// SIMATIC S7-200 project (STEP 7-Micro/WIN), CPU 221 REL 01.10

SYMBOL_TABLE USER1
S_tar            I0.0
S_top            I0.1
Den_1            Q0.0
Den_2            Q0.1
Den_3            Q0.2
Den_4            Q0.3
Den_5            Q0.4
END_SYMBOL_TABLE

ORGANIZATION_BLOCK MAIN:OB1
TITLE=PROGRAM COMMENTS
BEGIN
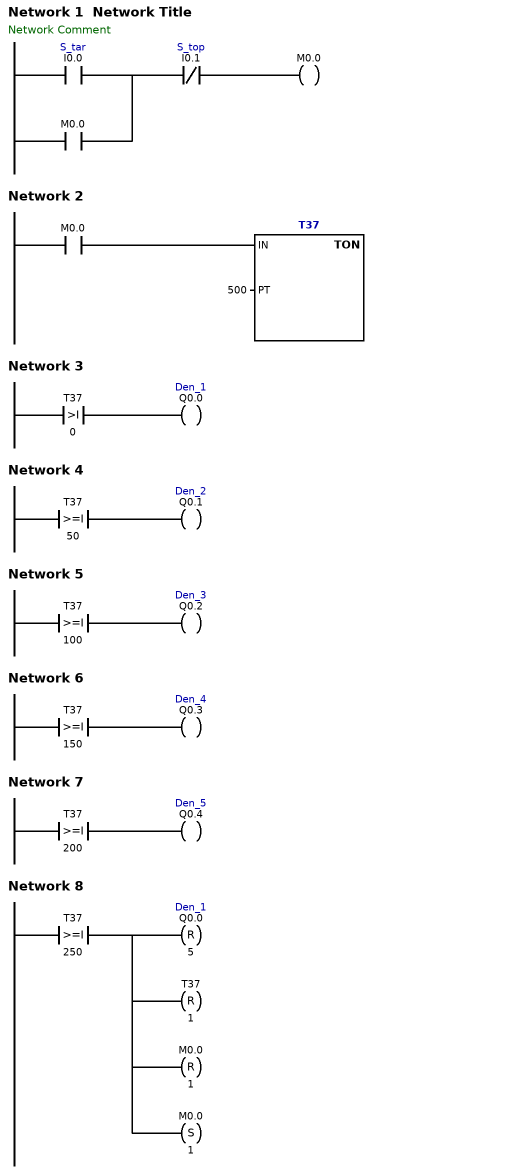
Network 1 // Network Title
// Network Comment
LD     S_tar:I0.0
O      M0.0
AN     S_top:I0.1
=      M0.0
Network 2
LD     M0.0
TON    T37, 500
Network 3
LDW>   T37, 0
=      Den_1:Q0.0
Network 4
LDW>=  T37, 50
=      Den_2:Q0.1
Network 5
LDW>=  T37, 100
=      Den_3:Q0.2
Network 6
LDW>=  T37, 150
=      Den_4:Q0.3
Network 7
LDW>=  T37, 200
=      Den_5:Q0.4
Network 8
LDW>=  T37, 250
R      Den_1:Q0.0, 5
R      T37, 1
R      M0.0, 1
S      M0.0, 1
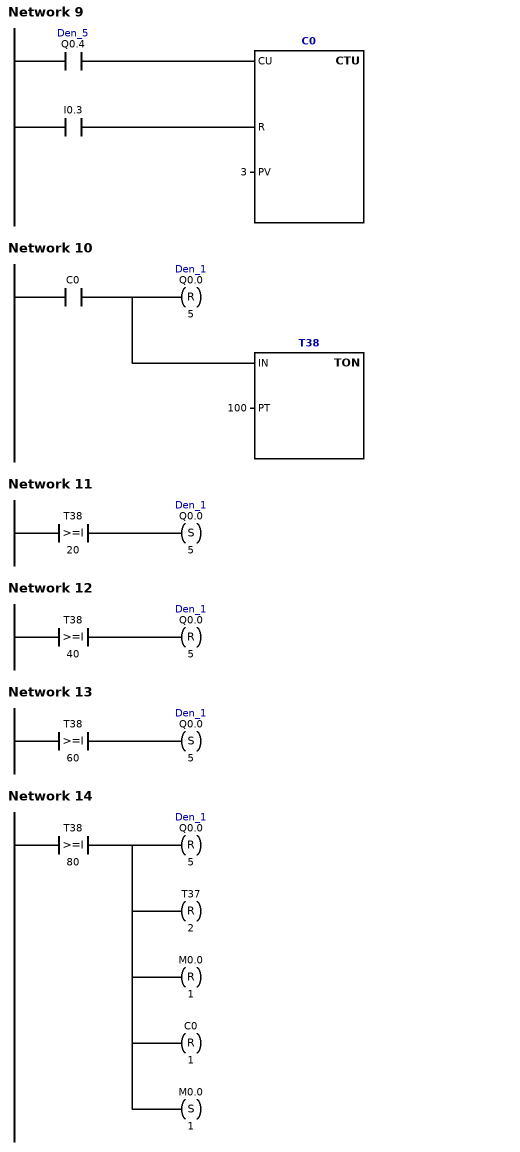
Network 9
LD     Den_5:Q0.4
LD     I0.3
CTU    C0, 3
Network 10
LD     C0
R      Den_1:Q0.0, 5
TON    T38, 100
Network 11
LDW>=  T38, 20
S      Den_1:Q0.0, 5
Network 12
LDW>=  T38, 40
R      Den_1:Q0.0, 5
Network 13
LDW>=  T38, 60
S      Den_1:Q0.0, 5
Network 14
LDW>=  T38, 80
R      Den_1:Q0.0, 5
R      T37, 2
R      M0.0, 1
R      C0, 1
S      M0.0, 1
END_ORGANIZATION_BLOCK
